GLOBALCONSTANTS DefaultPool_Joystick_Numeric (* Numeric object pool constants (ID, Scale, Offset, Decimals) *)
  PACKAGE Uebungen::const::UT::Joystick;
END_GLOBALCONSTANTS
